SUBAPPLICATION Uebung_170_AX (* Exercise for AX_D_FF *)
  (* Standard: 61499-2; Description: Copyright (c) 2025 Meisterschulen am Ostbahnhof This program and the accompanying materials are made available under the terms of the Eclipse Public License 2.0 which is available at https://www.eclipse.org/legal/epl-2.0/ SPDX-License-Identifier: EPL-2.0 *)
  (* Version 1.0, 2025-02-01, Franz Höpfinger, Meisterschulen am Ostbahnhof *)
  PACKAGE Uebungen;
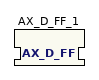
  FBS
    AX_D_FF_1 : adapter::events::unidirectional::AX_D_FF;
  END_FBS
END_SUBAPPLICATION
